// TIA Portal project "FC Programming" (V15.1)

(* hardware
DEVICE "S71500/ET200MP station_1"  S7-1500 station
   slot 0: "Rail_0"  Rack  6ES7 590-1***0-0AA0
   slot 0: "PM 190W 120/230VAC"  PM 190W 120/230VAC  6EP1333-4BA00
   slot 1: "PLC_1"  CPU 1516-3 PN/DP  6ES7 516-3AN01-0AB0  V2.6
      slot 3: "CPU display_1"  6ES7591-1BA00-0AA0
   slot 2: "DQ 32x24VDC/0.5A HF_1"  DQ 32x24VDC/0.5A HF  6ES7 522-1BL01-0AB0  V1.1
   slot 3: "DI 32x24VDC HF_1"  DI 32x24VDC HF  6ES7 521-1BL00-0AB0  V2.1
   slot 4: "AQ 4xU/I ST_1"  AQ 4xU/I ST  6ES7 532-5HD00-0AB0  V2.2
   slot 5: "AI 8xU/I/RTD/TC ST_1"  AI 8xU/I/RTD/TC ST  6ES7 531-7KF00-0AB0  V2.2
*)

// ===== PLC "PLC_1"  CPU 1516-3 PN/DP =====

VAR_GLOBAL   // PLC tag table "Full_Tag_Table"
   "Panel Emergency Stop" AT %I2.7 : Bool;
   "Start switch" AT %I0.2 : Bool;
   "Stop switch" AT %I0.3 : Bool;
   "Sort area IR" AT %I0.4 : Bool;
   "Sort Area Inductive" AT %I0.5 : Bool;
   "Sort Solenoid Sensor" AT %I0.6 : Bool;
   "Assembly Chute IR" AT %I0.7 : Bool;
   "Assembly Area Through Beam" AT %I1.1 : Bool;
   "Assembly Area Capacitor" AT %I1.2 : Bool;
   "Assembly Area Inductive" AT %I1.3 : Bool;
   "Reject Area IR" AT %I1.4 : Bool;
   "Reject Solenoid Sensor" AT %I1.5 : Bool;
   "Oven Through Beam" AT %I1.6 : Bool;
   "Loading Area Inductive" AT %I1.7 : Bool;
   "Chain Conveyor" AT %Q0.0 : Bool;
   "Sort Solenoid" AT %Q0.1 : Bool;
   "Reject Solenoid" AT %Q0.2 : Bool;
   "Rotary Solenoid" AT %Q0.3 : Bool;
   "Belt Conveyor Direction" AT %Q0.4 : Bool;
   "System Run_Green Lamp" AT %Q3.0 : Bool;
   "Sysyem Stop_Red Lamp" AT %Q3.2 : Bool;
   "Emergency stop" AT %I1.0 : Bool;
   "Ring Queue counter Full" AT %M4.0 : Bool;
   "Sort Solenoid error" AT %M4.3 : Bool;
   "Counter value" AT %MW0 : Int;
   "Reject Solenoid Error" AT %M4.7 : Bool;
   "HMI_Start" AT %M4.1 : Bool;
   "HMI_Stop" AT %M4.2 : Bool;
   "Counter Reset" AT %M4.4 : Bool;
END_VAR

FUNCTION "Conveyors_MANUAL" : Void   // FC1, LAD
TITLE = Motor control in manual mode
{ S7_Optimized_Access := 'TRUE' }
VERSION : 0.1
   VAR_INPUT
      "Start switch" : Bool;
      "Emergency stop" : Bool;
      "Panel emergency stop" : Bool;
   END_VAR
   VAR_OUTPUT
      "Chain Conveyor" : Bool;
      "Belt Conveyor" : Bool;
   END_VAR
   VAR_TEMP
      "Manual enable OK" : Bool;
   END_VAR
BEGIN

REGION Network 1: Manual enable ok
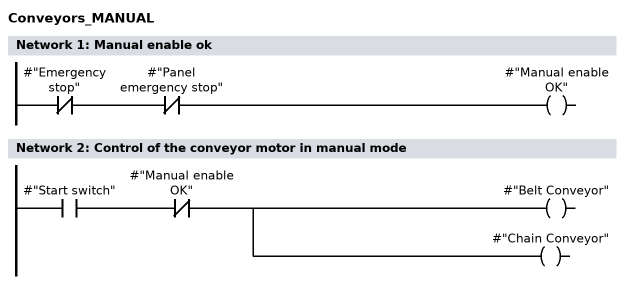
   RUNG wire#powerrail
      I_Contact( #"Emergency stop" )
      I_Contact( #"Panel emergency stop" )
      Coil( #"Manual enable OK" )
   END_RUNG
   // the same network as SCL:
   #"Manual enable OK" := NOT #"Emergency stop" AND NOT #"Panel emergency stop";
END_REGION

REGION Network 2: Control of the conveyor motor in manual mode
   RUNG wire#powerrail
      Contact( #"Start switch" )
      I_Contact( #"Manual enable OK" )
      wire#w1
      Coil( #"Belt Conveyor" )
   END_RUNG
   RUNG wire#w1
      Coil( #"Chain Conveyor" )
   END_RUNG
   // the same network as SCL:
   #"Belt Conveyor" := #"Start switch" AND NOT #"Manual enable OK";
   #"Chain Conveyor" := #"Belt Conveyor";
END_REGION
END_FUNCTION

ORGANIZATION_BLOCK "Main"   // OB1, LAD, ProgramCycle
TITLE = "Main Program Sweep (Cycle)"
{ S7_Optimized_Access := 'TRUE' }
VERSION : 0.1
   VAR_INPUT
      Initial_Call : Bool;   // Initial call of this OB
      Remanence : Bool;   // =True, if remanent data are available
   END_VAR
BEGIN

REGION Network 1
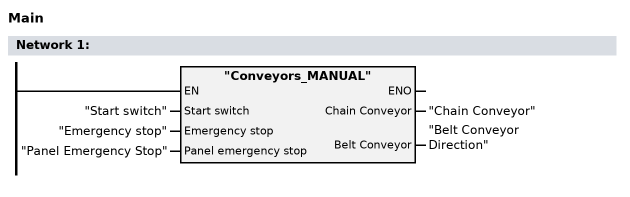
   RUNG wire#powerrail
      "Conveyors_MANUAL"("Start switch" := "Start switch", "Emergency stop" := "Emergency stop", "Panel emergency stop" := "Panel Emergency Stop", "Chain Conveyor" => "Chain Conveyor", "Belt Conveyor" => "Belt Conveyor Direction")
   END_RUNG
   // the same network as SCL:
   "Conveyors_MANUAL"("Start switch" := "Start switch",
                      "Emergency stop" := "Emergency stop",
                      "Panel emergency stop" := "Panel Emergency Stop",
                      "Chain Conveyor" => "Chain Conveyor",
                      "Belt Conveyor" => "Belt Conveyor Direction");
END_REGION
END_ORGANIZATION_BLOCK